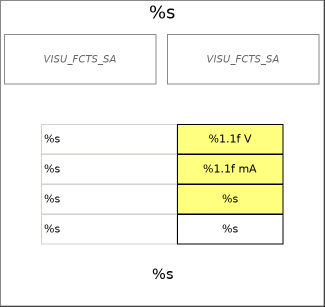
VISUALIZATION SA_EFFLUVAGE  // 325x307
VAR_IN_OUT
	m_input_effluvage:		BLOCK_PRG_EFFLUVAGE;
	m_Input_Machine:		BLOCK_MODE_MARCHE_V2_0;
END_VAR
    RoundedRectangle (0,0 325x307), "%s", text list: 'TextList_Effluvage', text index: 1
    Frame (4,34 152x50)
        shows VISU_FCTS_SA(m_Input_ID_XML := 29, m_Input_Operation := m_input_effluvage.Effluvage.OP_Marche_Eff, m_Input_UserRight := PRG_USER.ACTU_USER.FONCTION_SA)
    Frame (167,34 152x50)
        shows VISU_FCTS_SA(m_Input_ID_XML := 7, m_Input_Operation := m_input_effluvage.Effluvage.OP_Arret_Eff, m_Input_UserRight := PRG_USER.ACTU_USER.FONCTION_SA)
    Textfield (41,154 136x30), "%s", text list: 'TextList_Effluvage', text index: 2
    Textfield (41,184 136x30), "%s", text list: 'TextList_Effluvage', text index: 3
    Rectangle (177,154 106x30), "%1.1f mA", text variable: m_input_effluvage.Effluvage.PRM_consigne, input disabled if: (NOT PRG_User.ACTU_USER.MAINTENANCE AND NOT PRG_User.ACTU_USER.FONCTION_SA AND NOT PRG_User.ACTU_USER.MODIF_ENLIGNE) OR (NOT MACHINE.STATE_Wait_Prod AND NOT MACHINE.STATE_Manu)
        OnMouseClick: write the text variable via InputWithLimits, min 0
    Rectangle (177,184 106x30), "%s", text variable: m_input_effluvage.Effluvage.PRM_TPS_effluvage, input disabled if: (NOT PRG_User.ACTU_USER.MAINTENANCE AND NOT PRG_User.ACTU_USER.FONCTION_SA AND NOT PRG_User.ACTU_USER.MODIF_ENLIGNE) OR (NOT MACHINE.STATE_Wait_Prod AND NOT MACHINE.STATE_Manu)
        OnMouseClick: write the text variable via InputWithLimits, min 0
    Textfield (41,214 136x30), "%s", text list: 'TextList_Effluvage', text index: 4
    Rectangle (177,214 106x30), "%s", text variable: m_input_effluvage.Effluvage.TIMER_Effluvage.ET, input disabled if: (NOT PRG_User.ACTU_USER.MAINTENANCE AND NOT PRG_User.ACTU_USER.FONCTION_SA AND NOT PRG_User.ACTU_USER.MODIF_ENLIGNE) OR (NOT MACHINE.STATE_Wait_Prod AND NOT MACHINE.STATE_Manu)
    Rectangle (42,259 242x30), "%s", text variable: PRG_EFFLUVAGE.Effluvage.TIMER_Effluvage.ET, invisible if: Not PRG_EFFLUVAGE.Effluvage.OP_Marche_Eff.Etape.3, text list: 'TextList_Gaz', text index: 4
    Textfield (41,124 136x30), "%s", text list: 'TextList_Effluvage', text index: 5
    Rectangle (177,124 106x30), "%1.1f V", text variable: m_input_effluvage.Effluvage.PRM_Tension_attendue, input disabled if: (NOT PRG_User.ACTU_USER.MAINTENANCE AND NOT PRG_User.ACTU_USER.FONCTION_SA AND NOT PRG_User.ACTU_USER.MODIF_ENLIGNE) OR (NOT MACHINE.STATE_Wait_Prod AND NOT MACHINE.STATE_Manu)
        OnMouseClick: write the text variable via InputWithLimits, min 0
END_VISUALIZATION

(* stored: Version 1.1.0.1, ProductVersion 3.1.4024.11
   Visu SA_EFFLUVAGE: Id {b229d817-db48-486e-8b2f-db036de5ed2a} *)
